Yaskawa INFORM job: R1_W18,19,21(0,0)_KM-OKNEW_MP.JBI

/JOB
//NAME R1_W18,19,21(0,0)_KM-OKNEW_MP
///FOLDERNAME KRIS-SCIANA
//POS
///NPOS 88,88,0,5,0,0
///TOOL 0
///POSTYPE PULSE
///PULSE
C00000=-165945,-65747,-78398,-11730,94813,86069
C00001=-225738,-29129,-36820,-61092,45172,49948
C00002=-227041,-26413,-34946,-60254,44485,49501
C00003=-227207,-24592,-33670,-60039,44458,49378
C00004=-237456,-39019,-43586,-39021,28175,39239
C00005=-237530,-37534,-42645,-38724,28284,39091
C00006=-238362,-37606,-42693,-37740,27911,38632
C00007=-236638,-41709,-45274,-40385,28277,39894
C00008=-227197,-30656,-28257,-80893,39459,56892
C00009=-224091,-34376,-30000,-82400,41545,57754
C00010=-225738,-29129,-36820,-61092,45172,49948
C00011=-225738,-27920,-28129,-65451,42941,52685
C00012=-226983,-26160,-26909,-64802,42194,52319
C00013=-227202,-23846,-25282,-64524,42136,52156
C00014=-233227,-34794,-32737,-55973,30656,47784
C00015=-233341,-32754,-31394,-55574,30716,47580
C00016=-234428,-32958,-31529,-54757,30061,47174
C00017=-233341,-32754,-31394,-55574,30716,47580
C00018=-230699,-46358,-39944,-59876,31369,49797
C00019=-220936,-55036,-44073,-77006,39978,56936
C00020=-200682,-58218,-45802,-80292,54272,59368
C00021=-209639,-77270,-46477,-91612,78281,60493
C00022=178105,-72497,-44360,72515,40978,-24705
C00023=157900,67762,47803,76590,91490,-60139
C00024=160086,65038,44626,76467,90101,-59697
C00025=161508,64015,43441,76361,89159,-59481
C00026=161799,64427,43919,76335,88934,-59492
C00027=162551,28740,5640,71968,73206,-54657
C00028=163088,29659,6548,71873,72813,-54633
C00029=163408,28210,5119,71765,72642,-54534
C00030=161799,27490,4415,72104,73749,-54692
C00031=159860,62185,50950,86211,89235,-60844
C00032=160086,65038,44626,76467,90101,-59697
C00033=160567,66393,59893,76368,87465,-63546
C00034=161462,67229,60876,76403,86788,-63544
C00035=162034,68792,62724,76418,86297,-63641
C00036=161811,43273,34062,75782,77522,-60316
C00037=162300,44246,35097,75781,77142,-60332
C00038=162605,42812,33575,75722,76982,-60214
C00039=162300,44246,35097,75781,77142,-60332
C00040=157211,46506,37518,76082,80632,-60954
C00041=157670,65355,55356,86172,90720,-61418
C00042=161021,60847,32788,71661,91289,-58028
C00043=158071,42272,26850,85179,79726,-64183
C00044=160900,49335,52274,105567,79047,-73988
C00045=160407,59632,31901,71739,91677,-58132
C00046=160676,63082,35844,71667,91272,-58387
C00047=160929,49148,52068,105566,79020,-73978
C00048=160722,49177,52101,105542,79169,-73963
C00049=161225,48151,50953,105572,78773,-73921
C00050=160473,59253,70129,101537,81612,-81824
C00051=156183,50855,46384,99936,83176,-76860
C00052=151897,58426,66630,87129,82620,-71919
C00053=158751,51722,59033,87847,77807,-71164
C00054=160151,49894,57005,87950,76824,-70983
C00055=160407,59632,31901,71739,91677,-58132
C00056=160676,63082,35844,71667,91272,-58387
C00057=160214,47789,52341,87573,76909,-70139
C00058=151932,45808,25021,85459,84488,-63059
C00059=157434,41112,20051,84712,80618,-62540
C00060=160135,39734,18896,84350,78685,-62423
C00061=160407,59632,31901,71739,91677,-58132
C00062=160676,63082,35844,71667,91272,-58387
C00063=160165,50037,57157,87955,76814,-70996
C00064=156942,58566,66790,87841,79014,-71800
C00065=148876,27456,33542,86429,85194,-69951
C00066=224712,-65391,-70566,-27443,33176,35029
C00067=213770,-36542,-34460,77474,7084,-9175
C00068=217029,-28962,-25359,165424,2563,-53091
C00069=226738,-22872,-44138,-26151,38823,34122
C00070=225474,-24610,-45368,-24938,38325,33575
C00071=216815,-28472,-25029,161687,2573,-51425
C00072=216758,-28579,-25093,160911,2599,-51077
C00073=216562,-28626,-25134,158061,2661,-49812
C00074=216446,-27954,-24673,155770,2644,-48789
C00075=216538,-28216,-23367,164106,3479,-52503
C00076=216650,-37317,-29390,169486,4387,-54899
C00077=214272,-33613,-26176,108147,6753,-22913
C00078=214465,-33157,-25875,108062,6602,-22875
C00079=214164,-33211,-25911,107599,6817,-22666
C00080=214140,-14416,19283,164946,20973,-48668
C00081=217554,-35080,-3939,169426,16769,-50400
C00082=215729,-48765,-65733,21008,15669,16203
C00083=214258,-35470,-56996,22810,17401,15515
C00084=214189,-33167,-25881,107603,6800,-22674
C00085=218232,-57197,-39676,150711,6696,-41886
C00086=106022,-135537,-66235,115408,55550,-32403
C00087=10106,-66575,-39760,6607,87446,-74437
BC00000=342908,239,1075157
BC00001=398174,15,1075175
BC00002=398174,15,1075175
BC00003=398174,15,1075175
BC00004=398174,15,1075175
BC00005=398174,15,1075175
BC00006=398174,15,1075175
BC00007=398174,15,1075175
BC00008=398174,15,1075175
BC00009=398174,15,1075175
BC00010=398174,15,1075175
BC00011=398174,15,694659
BC00012=398174,15,694659
BC00013=398174,15,694659
BC00014=398174,15,694659
BC00015=398174,15,694659
BC00016=398174,15,694659
BC00017=398174,15,694659
BC00018=398174,15,694659
BC00019=398174,15,890503
BC00020=398174,15,890503
BC00021=394883,45674,1071776
BC00022=394883,231390,1071776
BC00023=365912,447627,1041849
BC00024=365912,447627,1041849
BC00025=365912,447627,1041849
BC00026=365912,447627,1041849
BC00027=365912,447627,1041849
BC00028=365912,447627,1041849
BC00029=365912,447627,1041849
BC00030=365912,447627,1041849
BC00031=365912,447627,1041849
BC00032=365912,447627,1041849
BC00033=365912,447627,693708
BC00034=365912,447627,693708
BC00035=365911,447627,693705
BC00036=365912,447627,693708
BC00037=365912,447627,693708
BC00038=365912,447627,693708
BC00039=365912,447627,693708
BC00040=365912,447627,693708
BC00041=365912,447627,1041849
BC00042=368384,441548,1075175
BC00043=360608,449199,1075175
BC00044=360608,449199,1075175
BC00045=360608,449199,1075175
BC00046=360608,449199,1075175
BC00047=360608,449199,894365
BC00048=360608,449199,731682
BC00049=360608,449199,597180
BC00050=360608,449199,610410
BC00051=360608,449199,610410
BC00052=360608,449199,871920
BC00053=360608,449199,871920
BC00054=360608,449199,871920
BC00055=360608,449199,1075175
BC00056=360608,449199,1075175
BC00057=360608,449199,655426
BC00058=360609,449199,890554
BC00059=360609,449199,890554
BC00060=360608,449199,890556
BC00061=360608,449199,1075175
BC00062=360608,449199,1075175
BC00063=360608,449199,871921
BC00064=360608,449199,871921
BC00065=360608,408502,871921
BC00066=398174,68400,1075175
BC00067=398174,60897,1075175
BC00068=398174,60897,1072583
BC00069=398174,60897,1075175
BC00070=398174,60897,1075175
BC00071=398174,60897,895364
BC00072=398174,60897,751044
BC00073=398174,60897,648257
BC00074=398174,60897,542662
BC00075=398099,60897,542662
BC00076=398099,60897,542662
BC00077=398174,60897,775711
BC00078=392644,57641,759002
BC00079=392644,57641,759001
BC00080=392644,57641,759002
BC00081=392644,57641,759002
BC00082=392644,57641,759002
BC00083=392644,57641,759002
BC00084=392644,57641,759002
BC00085=392644,57641,759002
BC00086=392644,373033,759002
BC00087=221411,449199,1015609
///POSTYPE BASE
///RECTAN
///RCONF 0,0,0,0,1,0,0,0,0,0,0,0,0,0,0,0,0,0,0,0,0,0,0,0
P00006=2.006,1.622,-0.565,0.0000,0.0000,0.0000
///RCONF 0,0,0,0,0,0,0,0,0,0,0,0,0,0,0,0,0,0,0,0,0,0,0,0
P00026=2.644,0.055,-2.583,0.0000,0.0000,0.0000
P00027=2.278,0.099,-4.210,0.0000,0.0000,0.0000
P00028=-1.778,-0.182,-2.050,0.0000,0.0000,0.0000
P00029=1.749,4.006,-0.261,0.0000,0.0000,0.0000
//INST
///DATE 2025/04/18 08:23
///ATTR SC,RW
///GROUP1 RB1,BS1
NOP
SFTOF
MOVJ C00000 BC00000 VJ=100.00
MOVL C00001 BC00001 V=500.0
MOVL C00002 BC00002 V=60.0
REFP 3 C00003 BC00003
CALL JOB:SEARCH-R1
SET P027 P006
SFTON P027
MOVL C00004 BC00004 V=60.0
MOVL C00005 BC00005 V=60.0
REFP 3 C00006 BC00006
CALL JOB:SEARCH-R1
SET P027 P006
SFTON P027
MOVL C00007 BC00007 V=60.0
MOVL C00008 BC00008 V=166.7
MOVL C00009 BC00009 V=166.7
'DOL
MOVL C00010 BC00010 V=166.7
MOVL C00011 BC00011 V=166.7
MOVL C00012 BC00012 V=60.0
REFP 3 C00013 BC00013
CALL JOB:SEARCH-R1
SET P029 P006
SFTON P029
MOVL C00014 BC00014 V=60.0
MOVL C00015 BC00015 V=60.0
REFP 3 C00016 BC00016
CALL JOB:SEARCH-R1
SET P029 P006
SFTON P029
MOVL C00017 BC00017 V=60.0
MOVL C00018 BC00018 V=60.0
MOVL C00019 BC00019 V=166.7
MOVL C00020 BC00020 V=166.7
SFTOF
'DRUGA STRONA
MOVJ C00021 BC00021 VJ=40.00
MOVJ C00022 BC00022 VJ=60.00
MOVL C00023 BC00023 V=333.3
MOVL C00024 BC00024 V=166.7
MOVL C00025 BC00025 V=60.0
REFP 3 C00026 BC00026
CALL JOB:SEARCH-R1
SET P026 P006
SFTON P026
MOVL C00027 BC00027 V=60.0
MOVL C00028 BC00028 V=60.0
REFP 3 C00029 BC00029
CALL JOB:SEARCH-R1
SET P026 P006
SFTON P026
MOVL C00030 BC00030 V=60.0
MOVL C00031 BC00031 V=100.0
'DOL
MOVL C00032 BC00032 V=166.7
MOVL C00033 BC00033 V=166.7
MOVL C00034 BC00034 V=60.0
REFP 3 C00035 BC00035
CALL JOB:SEARCH-R1
SET P028 P006
SFTON P028
MOVL C00036 BC00036 V=60.0
MOVL C00037 BC00037 V=60.0
REFP 3 C00038 BC00038
CALL JOB:SEARCH-R1
SET P028 P006
SFTON P028
MOVL C00039 BC00039 V=60.0
MOVL C00040 BC00040 V=100.0
MOVL C00041 BC00041 V=166.7
'Path S879 (for W18)
SFTOF
CALL JOB:COFNIJ_DRUT
SFTON P026
MOVL C00042 BC00042 V=333.3
MOVL C00043 BC00043 V=250.0
MOVL C00044 BC00044 V=166.7 PL=0
REFP 1 C00045 BC00045
REFP 2 C00046 BC00046
MACRO1 MJ#(0) ARGF6
ARCON
MOVL C00047 BC00047 V=13.3
MOVL C00048 BC00048 V=10.8
SFTON P028
MOVL C00049 BC00049 V=10.8
MOVL C00050 BC00050 V=10.8
ARCOF
'Path W883_C
SFTOF
MOVL C00051 BC00051 V=333.3
COMM SFTON P028
COMM MOVL C00052 BC00052 V=100.0
COMM MOVL C00053 BC00053 V=100.0
COMM MOVL C00054 BC00054 V=100.0 PL=0
COMM REFP 1 C00055 BC00055
COMM REFP 2 C00056 BC00056
COMM MACRO1 MJ#(0) ARGF6
COMM ARCON
COMM MOVL C00057 BC00057 V=13.3
COMM ARCOF
COMM 'Path W883_B
COMM SFTOF
COMM SFTON P028
COMM MOVL C00058 BC00058 V=100.0
COMM MOVL C00059 BC00059 V=100.0
COMM MOVL C00060 BC00060 V=100.0 PL=0
COMM REFP 1 C00061 BC00061
COMM REFP 2 C00062 BC00062
COMM MACRO1 MJ#(0) ARGF6
COMM ARCON
COMM SFTON P028
COMM MOVL C00063 BC00063 V=13.3
COMM ARCOF
COMM MOVL C00064 BC00064 V=100.0
SFTOF
MOVL C00065 BC00065 V=100.0
MOVL C00066 BC00066 V=333.3
MOVL C00067 BC00067 V=166.7
SFTON P027
MOVL C00068 BC00068 V=100.0 PL=0
REFP 1 C00069 BC00069
REFP 2 C00070 BC00070
MACRO1 MJ#(0) ARGF6
ARCON
MOVL C00071 BC00071 V=10.8
MOVL C00072 BC00072 V=10.8
SFTON P029
MOVL C00073 BC00073 V=10.8
MOVL C00074 BC00074 V=10.8
MOVL C00075 BC00075 V=10.8
ARCOF
MOVL C00076 BC00076 V=166.7
SFTOF
COMM MOVJ C00077 BC00077 VJ=100.00
COMM SFTON P029
COMM MOVJ C00078 BC00078 VJ=100.00
COMM MACRO1 MJ#(0) ARGF6
COMM MOVL C00079 BC00079 V=50.0 PL=0
COMM ARCON
COMM MOVL C00080 BC00080 V=12.5
COMM ARCOF
COMM TIMER T=1.00
COMM SFTOF
COMM MOVJ C00081 BC00081 VJ=100.00
COMM MOVJ C00082 BC00082 VJ=25.00
COMM SFTON P029
COMM MOVJ C00083 BC00083 VJ=100.00 PL=0
COMM ARCON
COMM MOVL C00084 BC00084 V=12.5
COMM ARCOF
COMM TIMER T=1.00
COMM SFTOF
COMM MOVL C00085 BC00085 V=166.7
SFTOF
MOVJ C00086 BC00086 VJ=100.00
MOVJ C00087 BC00087 VJ=100.00
END
